Yaskawa INFORM job: TATCALIBRATE.JBI

/JOB
//NAME TATCALIBRATE
//POS
///NPOS 5,0,0,0,0,0
///TOOL 0
///POSTYPE PULSE
///PULSE
C00000=-7969,21694,-5134,1465,-52599,3149
C00001=-43487,10808,-30891,5060,-37212,17750
C00002=-24167,57720,22702,2808,-52785,10258
C00003=23516,61116,27250,-1344,-54873,-10642
C00004=42600,11752,-30041,-3542,-38135,-18280
//INST
///DATE 2026/04/27 19:13
///ATTR SC,RW
///GROUP1 RB1
NOP
MOVJ C00000 VJ=0.78
MOVJ C00001 VJ=0.78
MOVJ C00002 VJ=0.78
MOVJ C00003 VJ=0.78
MOVJ C00004 VJ=0.78
END
